INTERFACE I_Pump EXTENDS __SYSTEM.IQueryInterface

METHOD GetFlowRate : REAL
VAR_INPUT
END_VAR
END_METHOD

METHOD GetTotalVolume : REAL
VAR_INPUT
END_VAR
END_METHOD

METHOD Start : BOOL
VAR_INPUT
END_VAR
END_METHOD

METHOD Stop : BOOL
VAR_INPUT
END_VAR
END_METHOD

END_INTERFACE

(* stored: Version 1.1.0.1, ProductVersion 3.1.4024.16
   Itf I_Pump: Id {ea7fd118-907a-4da4-b0f0-ce22284fd583}
   Method GetFlowRate: Id {3263a391-b109-4005-91a9-10e115e5665b}
   Method GetTotalVolume: Id {7d729ab2-a39e-4bd5-a7c6-ea8d7a6128f0}
   Method Start: Id {23c5d9df-d554-4793-96f0-610c85052704}
   Method Stop: Id {14700fc8-b9d0-4692-a353-642995c1933e} *)
